PROGRAM z_TK1


(*-------------------------------------------------------------------------------------------------------*)
(*p150  Pre Aviso Manual Cubeta 1*)


(*-------------------------------------------------------------------------------------------------------*)


(*-------------------------------------------------------------------------------------------------------*)
(*v105  Ev. Vaciado con Bomba TK 1*)


(*-------------------------------------------------------------------------------------------------------*)
(*v106  Ev. Vaciado por Gravedad TK 1*)


(*-------------------------------------------------------------------------------------------------------*)
(*v50  Ev. Intro Rapida TK 1*)




(*-------------------------------------------------------------------------------------------------------*)
(*v51  Ev. Intro Lenta (Dosing) TK 1*)

(*-------------------------------------------------------------------------------------------------------*)
(*v103  Ev. Intercepta TK 1*)


(*-------------------------------------------------------------------------------------------------------*)
(*v101  Ev. Llenado TK 1*)


(*-------------------------------------------------------------------------------------------------------*)
(*v102  Ev. Retorno Maq -> TK 1*)

(*-------------------------------------------------------------------------------------------------------*)
(*v109  Ev. Mezcla TK 1*)

(*-------------------------------------------------------------------------------------------------------*)
(*v109  Ev. Vapor TK 1*)

END_PROGRAM

(* stored: Version 1.1.0.1, ProductVersion 3.1.4024.10
   POU z_TK1: Id {9b315c30-0982-4960-8aeb-bdb30ff2c6f4}, SpecialFunc None *)
